FUNCTION_BLOCK SPLIT_AL_INTO_AW (* this Function splits the 4 AW (WORD) adapters from a AL (LWORD) *)
  (* Standard: 61499-2; Description: Copyright (c) 2026 Meisterschulen am Ostbahnhof SPDX-License-Identifier: EPL-2.0 *)
  (* Version 1.0, 2026-05-16, Franz Höpfinger, Meisterschulen am Ostbahnhof, initial API and implementation and/or initial documentation *)
  PACKAGE adapter::splitting;
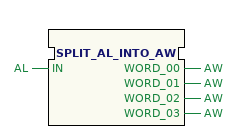
  SOCKETS
    IN : adapter::types::unidirectional::AL; (* LWORD Input *)
  END_SOCKETS
  PLUGS
    WORD_00 : adapter::types::unidirectional::AW; (* Word 0 *)
    WORD_01 : adapter::types::unidirectional::AW; (* Word 1 *)
    WORD_02 : adapter::types::unidirectional::AW; (* Word 2 *)
    WORD_03 : adapter::types::unidirectional::AW; (* Word 3 *)
  END_PLUGS
END_FUNCTION_BLOCK
